// TIA Portal V17 export
// export: Created 2023-04-03T06:31:42.1364756Z, ExportSetting WithDefaults, DisplayName Totally Integrated Automation Portal, DisplayVersion V17 Update 4, DisplayName TIA Portal Openness, DisplayVersion V17 Update 4, DisplayName TIA Portal Version Control Interface, DisplayVersion V17, DisplayName STEP 7 Professional, DisplayVersion V17 Update 4, DisplayName STEP 7 Safety, DisplayVersion V17, DisplayName WinCC Professional, DisplayVersion V17 Update 4
TYPE "W_PE_Block1"
// stored: IsFailsafeCompliant false
   STRUCT
      "G1.4_User_Psw" : Word;   // 1 / 40005
   END_STRUCT;
END_TYPE
